Staubli VAL3: aTcp.pgx

public program aTcp(point x_pUserTcp1, point x_pUserTcp2, point x_pUserTcp3, point x_pUserTcp4, bool& x_bCalcOk[], trsf& x_trUserTool[])
begin
  //-----------------------------------------------------------------------
  //Header begin
  //Description of program
  //  Same as aMainTcp except the points need to be already taught (no wizard)
  //  Caution : Defines only the X, Y, Z components of the TCP trsf
  //
  //Input parameters
  //  point x_pUserTcp1 to x_pUserTcp4
  //    role : 4 points used to calculates the TCP
  //    possible values : not applicable (taught points)
  //
  //Output parameters
  //  bool x_bCalcOk
  //    role : set to false if there is an error of calulation and true otherwise
  //  trsf x_trUserTool
  //    role : Contains settings tool (X, Y, Z)
  //History
  //  Creation : 07-04-08 - f.Rob
  //Header end
  //-----------------------------------------------------------------------

  //Initializing all parameters (trsf, point...)
  call valSetBack()

  call splitUp(x_pUserTcp1,x_pUserTcp2,x_pUserTcp3,x_pUserTcp4)
  call calculation(nS1[1],nS2[1],nS3[1],nS4[1],nS1[2],nS2[2],nS3[2],nS4[2],nS1[3],nS2[3],nS3[3],nS4[3])
  //If the tool calculation is not correct -> bAbort true
  x_bCalcOk=!bAbort
  if bAbort
    call valSetBack()
    x_trUserTool={0,0,0,0,0,0}
  else
    x_trUserTool={nToolX,nToolY,nToolZ,0,0,0}
  endIf
end
